Staubli VAL3: OnF2.pgx

program OnF2()
  local num l_ni
  local bool l_bRes
begin

  call setPoint(sItem)
  popUpMsg("选择点："+sItem)
end
